(* IEC 61131-3 sources: Lasal/CPU_5344_V01/Class/calcComplete, 1 file *)

(* ---- calcComplete.st ---- *)
(*!
<Class
	Name               = "calcComplete"
	Revision           = "0.0"
	RealtimeTask       = "false"
	CyclicTask         = "true"
	DefCyclictime      = "10 ms"
	BackgroundTask     = "false"
	DefBackground      = "10 ms"
	Sigmatek           = "false"
	OSInterface        = "false"
	HighPriority       = "false"
	Automatic          = "false"
	UpdateMode         = "Prescan"
	SharedCommandTable = "true"
	Objectsize         = "(284,120)">
	<Channels>
		<Server Name="calcDone" Visualized="true" Initialize="false" WriteProtected="false" Retentive="false"/>
		<Server Name="ClassSvr" Visualized="false" Initialize="false" WriteProtected="true" Retentive="false"/>
		<Server Name="elapsedTime" Visualized="false" Initialize="false" WriteProtected="true" Retentive="false"/>
		<Server Name="startCalc" Visualized="true" Initialize="false" WriteProtected="false" Retentive="false"/>
		<Server Name="stprCalc" Visualized="true" Initialize="false" WriteProtected="false" Retentive="false"/>
		<Client Name="ctrlCalc" Required="true" Internal="false"/>
		<Client Name="ctrlConvert" Required="true" Internal="false"/>
	</Channels>
</Class>
*)
calcComplete : CLASS
  //Servers:
	ClassSvr 	: SvrChCmd_DINT;
	stprCalc 	: SvrCh_DINT;
	startCalc 	: SvrCh_DINT;
	calcDone 	: SvrCh_DINT;
	elapsedTime 	: SvrCh_UDINT;
  //Clients:
	ctrlCalc 	: CltChCmd_calcOperationListV2;
	ctrlConvert 	: CltChCmd_convertOperationListToSLinesV2;
  //Variables:
		tmpTime 	: UDINT;
  //Functions:

	FUNCTION VIRTUAL GLOBAL CyWork
		VAR_INPUT
			EAX 	: UDINT;
		END_VAR
		VAR_OUTPUT
			state (EAX) 	: UDINT := READY;
		END_VAR;

	FUNCTION VIRTUAL GLOBAL startCalc::Write
		VAR_INPUT
			input (EAX) 	: DINT;
		END_VAR
		VAR_OUTPUT
			result (EAX) 	: DINT;
		END_VAR;
  //Tables:
	FUNCTION @STD
		VAR_OUTPUT
			ret_code	: CONFSTATES;
		END_VAR;
	FUNCTION GLOBAL TAB @CT_;
END_CLASS;

#pragma usingLtd calcOperationListV2
#pragma usingLtd convertOperationListToSLinesV2

//JdK 20-6-2019: calcComplete is created for 4284/Traffiroad / standard lib
// goal is to connect calcOperationList and convertOperationListToSLines

FUNCTION VIRTUAL GLOBAL calcComplete::startCalc::Write
	VAR_INPUT
		input (EAX) 	: DINT;
	END_VAR
	VAR_OUTPUT
		result (EAX) 	: DINT;
	END_VAR

	IF stprCalc=0 THEN
    calcDone:=-1;
    stprCalc:=1;
    tmpTime:=ops.tAbsolute;
    startCalc:= 1;
  ELSE
    startCalc:= 0;
  END_IF;
	result := startCalc;

END_FUNCTION

FUNCTION VIRTUAL GLOBAL calcComplete::CyWork
	VAR_INPUT
		EAX 	: UDINT;
	END_VAR
	VAR_OUTPUT
		state (EAX) 	: UDINT;(* := READY *)
	END_VAR

  CASE stprCalc OF

  0: //wait for start

  1: //start calculation
    IF ctrlCalc.stprCalc=0 THEN
      ctrlCalc.startCalc.Write(input:=1);
      IF ctrlCalc.calcDone= -1 THEN //means is started
        stprCalc+=2;
      END_IF;
    END_IF;

  3: //wait until calculation is done
    IF ctrlCalc.stprCalc=0 & ctrlCalc.calcDone>=0 THEN
      stprCalc+=1;
    ELSIF ctrlCalc.stprCalc=0 & ctrlCalc.calcDone=0 THEN
      stprCalc:= 0;
    END_IF;

  4: //start converting
    IF ctrlConvert.stprConvert=0 THEN
      ctrlConvert.startConvert.Write(input:=1);
      IF ctrlConvert.convertDone= -1 THEN //means is started
        stprCalc+=2;
      END_IF;
    END_IF;

  6: //wait until convertion is done
    IF ctrlConvert.stprConvert=0 & ctrlConvert.convertDone>=0 THEN
      stprCalc+=1;
    END_IF;

  7: //check if everything is ok
    IF ctrlCalc.calcDone=1 & ctrlConvert.convertDone=1 THEN
      calcDone:=1;
    ELSE
      calcDone:=0;
    END_IF;
    elapsedTime:=OPS.tAbsolute-tmpTime;
    stprCalc:=0;

  END_CASE;

END_FUNCTION
